{attribute 'GeneratedUsingTerminal: EL2262-0000-0004'}
{attribute addProperty BoxType "EL2262-0000-0004"}
{attribute addProperty Id "StartTimeNextOutputAT %I*UDINT4"}
{attribute addProperty CRC "579299316"}
{attribute addProperty Size "4"}
TYPE StartTimeNextOutput_228767F4 :
STRUCT
	{attribute addProperty Name "StartTimeNextOutput"}
	StartTimeNextOutput AT %I* : UDINT;
END_STRUCT
END_TYPE

(* stored: Version 1.2.0.0, ProductVersion 3.1.4024.9
   DUT StartTimeNextOutput_228767F4: Id {24022672-e759-435c-a319-cdbccc6ec230} *)
